(* IEC 61131-3 sources: plc_generation_empirical_study/datasets/task_bank_c06_reverse_bounded_runtime_v0_3/tasks/C06_V06_lean_composite/negative_control, 1 file *)

(* ---- NC1.st ---- *)
FUNCTION_BLOCK C06_V06_lean_composite
VAR_INPUT
    A_ChA : BOOL;
    A_ChB : BOOL;
    A_TestMode : BOOL;
    A_TestPermit : BOOL;
    A_ProcessRequest : BOOL;
    B_GoodPart : BOOL;
    B_RejectPart : BOOL;
    B_Reset : BOOL;
    B_BatchTarget : INT;
    B_RejectLimit : INT;
    SubsystemBEnable : BOOL;
    CrossReset : BOOL;
END_VAR
VAR_OUTPUT
    A_SafeEnable : BOOL;
    A_Disagree : BOOL;
    A_TestActive : BOOL;
    B_GoodCount : INT;
    B_RejectCount : INT;
    B_BatchDone : BOOL;
    B_QualityFault : BOOL;
    CrossReady : BOOL;
    CrossBlocked : BOOL;
END_VAR
VAR
    B_PrevGood : BOOL := FALSE;
    B_PrevReject : BOOL := FALSE;
END_VAR

A_Disagree := A_ChA <> A_ChB;
A_TestActive := A_TestMode AND A_TestPermit;
IF A_TestMode THEN
    A_SafeEnable := A_ProcessRequest AND A_TestPermit AND A_ChA;
ELSE
    A_SafeEnable := A_ProcessRequest AND A_ChA AND A_ChB;
END_IF;

IF CrossReset THEN
    CrossReady := FALSE;
ELSIF A_SafeEnable THEN
    CrossReady := TRUE;
END_IF;
CrossBlocked := FALSE;

IF SubsystemBEnable AND CrossReady THEN
    IF B_Reset THEN
        B_GoodCount := 0;
        B_RejectCount := 0;
        B_QualityFault := FALSE;
    ELSE
        IF B_RejectPart AND (NOT B_PrevReject) THEN
            B_RejectCount := B_RejectCount + 1;
        ELSIF B_GoodPart AND (NOT B_PrevGood) THEN
            B_GoodCount := B_GoodCount + 1;
        END_IF;
        IF B_RejectCount >= B_RejectLimit THEN
            B_QualityFault := TRUE;
        END_IF;
    END_IF;
    B_BatchDone := (B_GoodCount + B_RejectCount) >= B_BatchTarget;
    B_PrevGood := B_GoodPart;
    B_PrevReject := B_RejectPart;
ELSE
    B_GoodCount := 0;
    B_RejectCount := 0;
    B_BatchDone := FALSE;
    B_QualityFault := FALSE;
END_IF;

END_FUNCTION_BLOCK
